{attribute 'qualified_only'}
VAR_GLOBAL
	arrbySend_Data			: ARRAY [0..Sewts_TCP.MAX_QUEUE_SIZE] OF BYTE;
	arrbyReceive_Data		: ARRAY [0..Sewts_TCP.MAX_QUEUE_SIZE] OF BYTE;
END_VAR

(* stored: Version 1.1.0.1, ProductVersion 3.1.4024.12
   GVL GVX: Id {3c1176c5-fef7-4310-a5da-0b70b45f91be} *)
